// SIMATIC S7-200 project (STEP 7-Micro/WIN), CPU 221 REL 01.10

SYMBOL_TABLE USER1
Sen1             I0.0
sen2             I0.1
Sen3             I0.2
Sen4             I0.3
start            I0.4
estop            I0.5
m1               Q0.0
m2               Q0.1
cb               Q0.2
END_SYMBOL_TABLE

ORGANIZATION_BLOCK MAIN:OB1
TITLE=PROGRAM COMMENTS
BEGIN
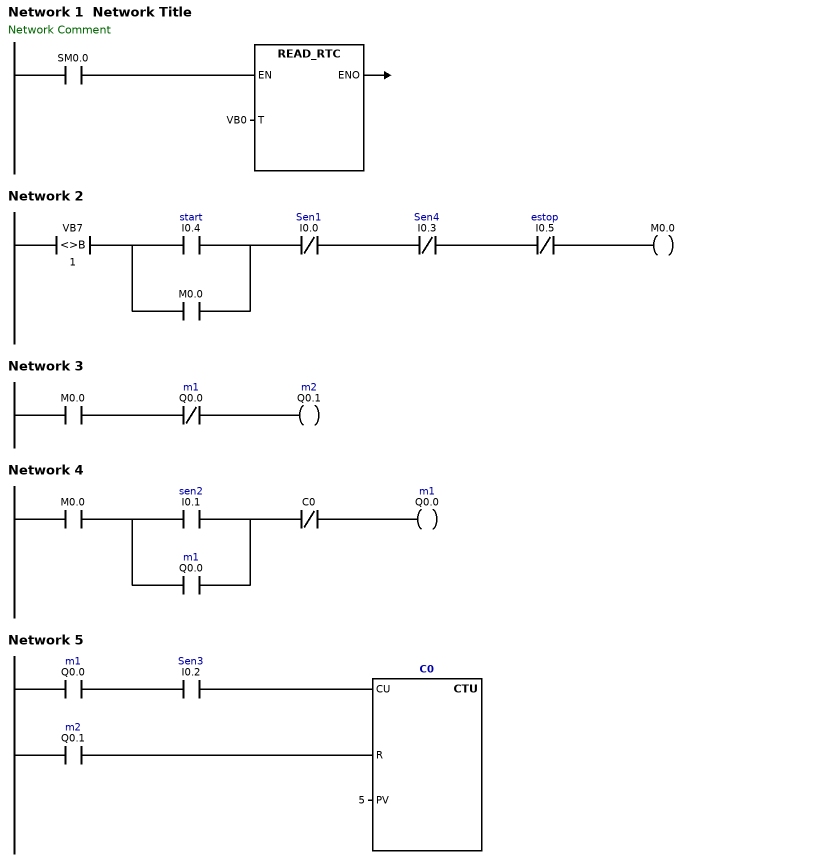
Network 1 // Network Title
// Network Comment
LD     SM0.0
TODR   VB0
Network 2
LDB<>  VB7, 1
LD     start:I0.4
O      M0.0
ALD
AN     Sen1:I0.0
AN     Sen4:I0.3
AN     estop:I0.5
=      M0.0
Network 3
LD     M0.0
AN     m1:Q0.0
=      m2:Q0.1
Network 4
LD     M0.0
LD     sen2:I0.1
O      m1:Q0.0
ALD
AN     C0
=      m1:Q0.0
Network 5
LD     m1:Q0.0
A      Sen3:I0.2
LD     m2:Q0.1
CTU    C0, 5
END_ORGANIZATION_BLOCK
